// Mitsubishi GX Works2 project: fenjian   PLC: FX3U/FX3UC

PROGRAM MAIN
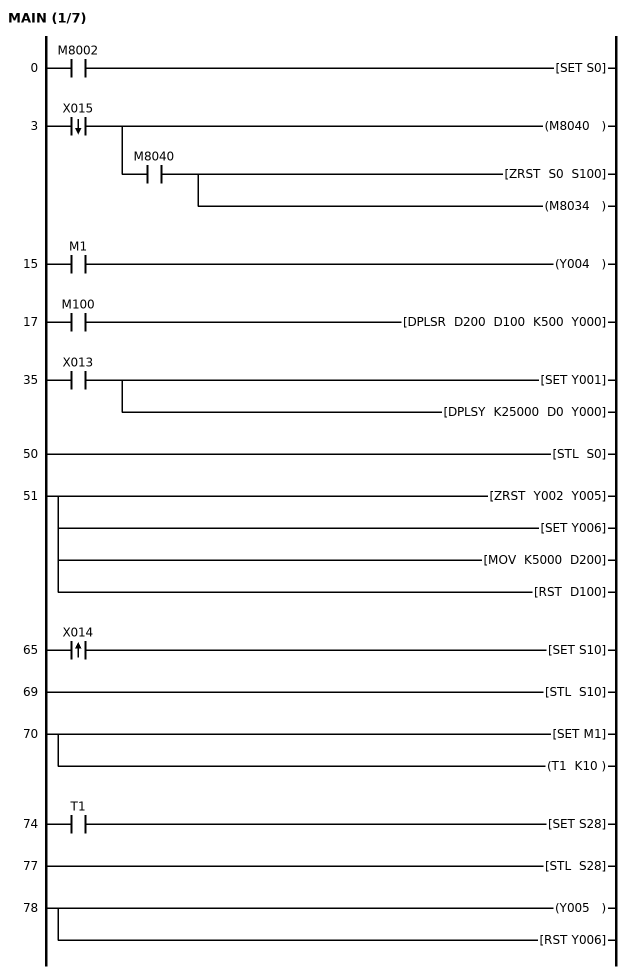
0     LD      M8002
      SET     S0
3     LDF     X015
      OUT     M8040
      AND     M8040
      ZRST    S0 S100
      OUT     M8034
15    LD      M1
      OUT     Y004
17    LD      M100
      DPLSR   D200 D100 K500 Y000
35    LD      X013
      SET     Y001
      DPLSY   K25000 D0 Y000
50    STL     S0
51    ZRST    Y002 Y005
      SET     Y006
      MOV     K5000 D200
      RST     D100
65    LDP     X014
      SET     S10
69    STL     S10
70    SET     M1
      OUT     T1 K10
74    LD      T1
      SET     S28
77    STL     S28
78    OUT     Y005
      RST     Y006
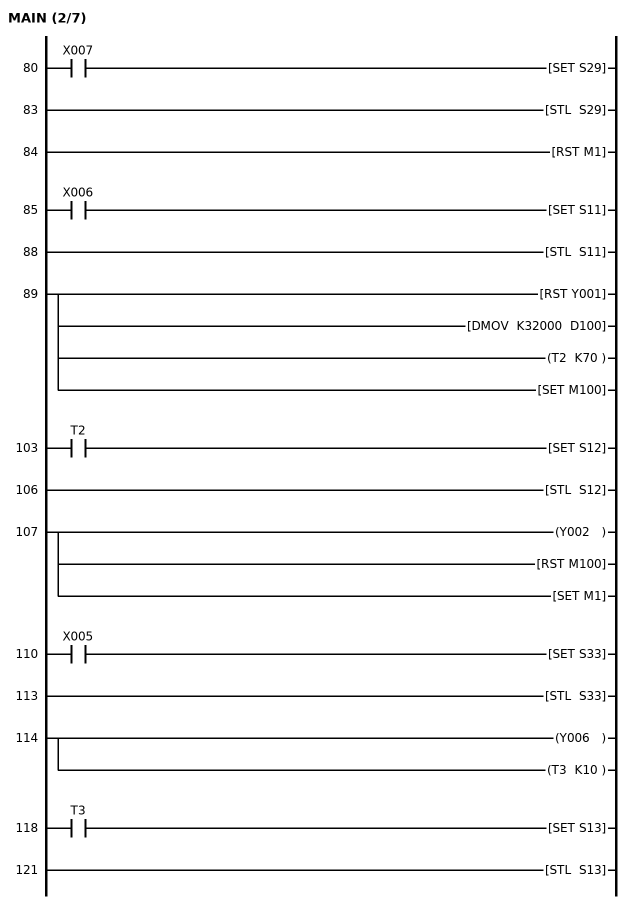
80    LD      X007
      SET     S29
83    STL     S29
84    RST     M1
85    LD      X006
      SET     S11
88    STL     S11
89    RST     Y001
      DMOV    K32000 D100
      OUT     T2 K70
      SET     M100
103   LD      T2
      SET     S12
106   STL     S12
107   OUT     Y002
      RST     M100
      SET     M1
110   LD      X005
      SET     S33
113   STL     S33
114   OUT     Y006
      OUT     T3 K10
118   LD      T3
      SET     S13
121   STL     S13
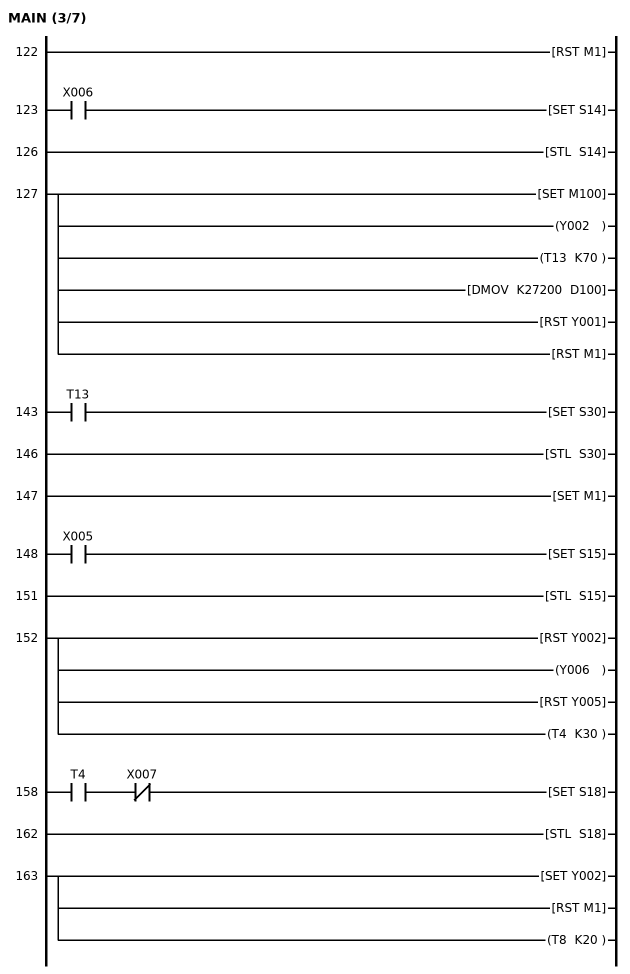
122   RST     M1
123   LD      X006
      SET     S14
126   STL     S14
127   SET     M100
      OUT     Y002
      OUT     T13 K70
      DMOV    K27200 D100
      RST     Y001
      RST     M1
143   LD      T13
      SET     S30
146   STL     S30
147   SET     M1
148   LD      X005
      SET     S15
151   STL     S15
152   RST     Y002
      OUT     Y006
      RST     Y005
      OUT     T4 K30
158   LD      T4
      ANI     X007
      SET     S18
162   STL     S18
163   SET     Y002
      RST     M1
      OUT     T8 K20
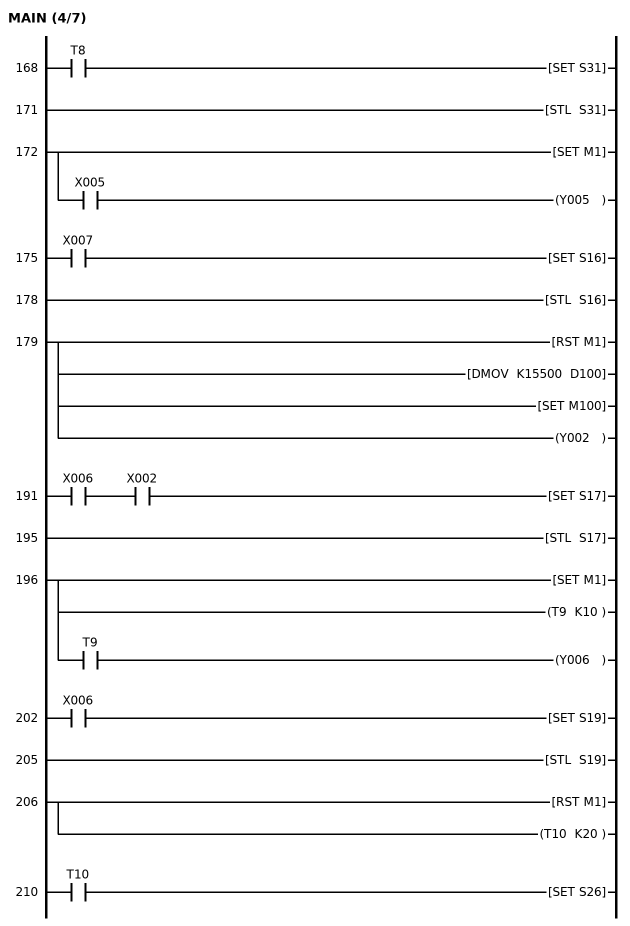
168   LD      T8
      SET     S31
171   STL     S31
172   SET     M1
      AND     X005
      OUT     Y005
175   LD      X007
      SET     S16
178   STL     S16
179   RST     M1
      DMOV    K15500 D100
      SET     M100
      OUT     Y002
191   LD      X006
      AND     X002
      SET     S17
195   STL     S17
196   SET     M1
      OUT     T9 K10
      AND     T9
      OUT     Y006
202   LD      X006
      SET     S19
205   STL     S19
206   RST     M1
      OUT     T10 K20
210   LD      T10
      SET     S26
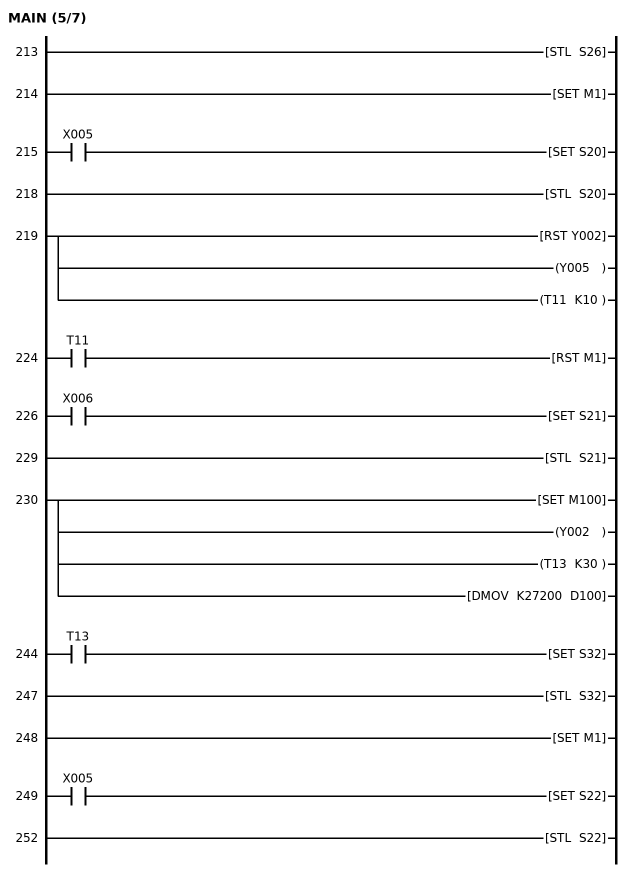
213   STL     S26
214   SET     M1
215   LD      X005
      SET     S20
218   STL     S20
219   RST     Y002
      OUT     Y005
      OUT     T11 K10
224   LD      T11
      RST     M1
226   LD      X006
      SET     S21
229   STL     S21
230   SET     M100
      OUT     Y002
      OUT     T13 K30
      DMOV    K27200 D100
244   LD      T13
      SET     S32
247   STL     S32
248   SET     M1
249   LD      X005
      SET     S22
252   STL     S22
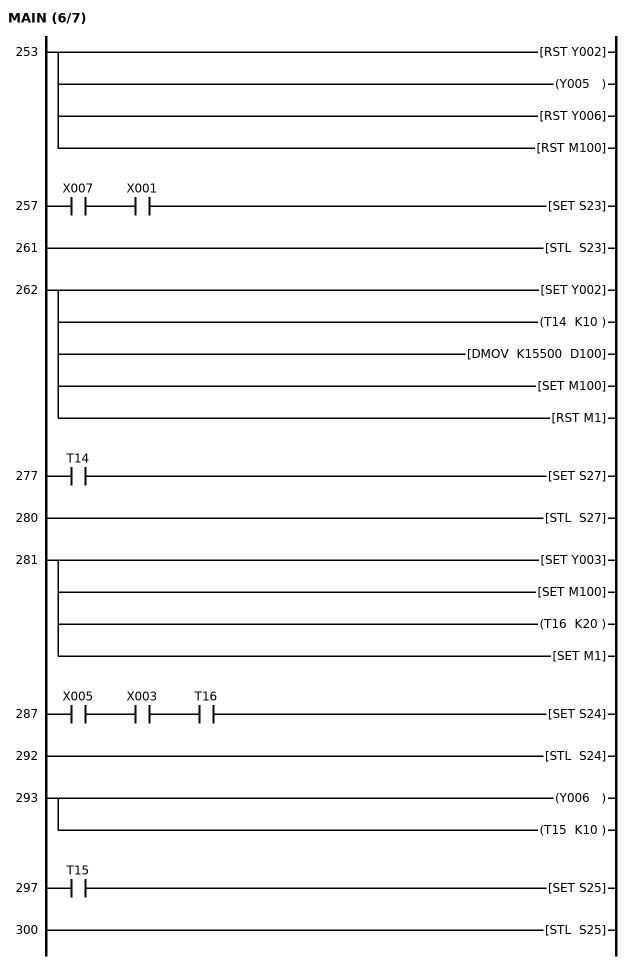
253   RST     Y002
      OUT     Y005
      RST     Y006
      RST     M100
257   LD      X007
      AND     X001
      SET     S23
261   STL     S23
262   SET     Y002
      OUT     T14 K10
      DMOV    K15500 D100
      SET     M100
      RST     M1
277   LD      T14
      SET     S27
280   STL     S27
281   SET     Y003
      SET     M100
      OUT     T16 K20
      SET     M1
287   LD      X005
      AND     X003
      AND     T16
      SET     S24
292   STL     S24
293   OUT     Y006
      OUT     T15 K10
297   LD      T15
      SET     S25
300   STL     S25
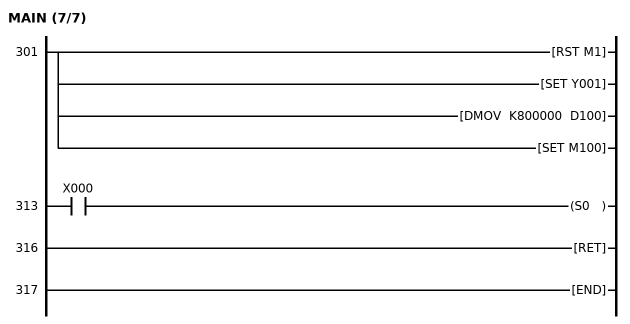
301   RST     M1
      SET     Y001
      DMOV    K800000 D100
      SET     M100
313   LD      X000
      OUT     S0
316   RET
317   END
END_PROGRAM

// device comments not shown above
BL1  ; 2
